// TIA Portal V21 export
VAR_GLOBAL   // PLC tag table "INSTRUMENTOS_ALARMES (ETA)"
   "NIVEL_MUITO_ALTO (ETA)" AT %M60.0 : Bool;
   "PRESSAO_ALTA (ETA)" AT %M60.1 : Bool;
END_VAR
